// TIA Portal V19 export
DATA_BLOCK "EnS_LAcycCom_ResourceManager"   // DB39
TITLE = Instance DB of LAcycCom ResourceManager Variant
// Instance DB of LAcycCom ResourceManager Variant
// stored: InstanceOfName LAcycCom_ResourceManager_Variant, InstanceOfType FB
"LAcycCom_ResourceManager_Variant"
   // VAR_INPUT
   //    enable : Bool;
   //    config : "LAcycCom_typeResourceManagerConf";
   // END_VAR
   // VAR_OUTPUT
   //    valid : Bool;
   //    busy : Bool;
   //    error : Bool;
   //    status : Word;
   //    diagnostics : "LAcycCom_typeResourceManagerDiag";
   // END_VAR
   // VAR_IN_OUT
   //    requestBufferHeader : "LAcycCom_typeRequestBufferHeader";
   //    requestBufferElements : Variant;
   // END_VAR
   // VAR
   //    statResourceAddInfo { ExternalAccessible := 'False'; ExternalVisible := 'False'; ExternalWritable := 'False'} : Array[0..9] of Struct
   //       IOSystem : Int;
   //       station : Int;
   //    END_STRUCT;
   //    instBufferLockWatchdog { ExternalAccessible := 'False'; ExternalVisible := 'False'; ExternalWritable := 'False'; S7_SetPoint := 'True'} : TON_TIME;
   //    instRuntime { ExternalAccessible := 'False'; ExternalVisible := 'False'; ExternalWritable := 'False'; S7_SetPoint := 'True'} : TON_TIME;
   //    instCycleTime { ExternalAccessible := 'False'; ExternalVisible := 'False'; ExternalWritable := 'False'; S7_SetPoint := 'True'} : TON_TIME;
   //    instGetIMData { ExternalAccessible := 'False'; ExternalVisible := 'False'; ExternalWritable := 'False'; S7_SetPoint := 'True'} : Get_IM_Data;
   //    statIM0Data { ExternalAccessible := 'False'; ExternalVisible := 'False'; ExternalWritable := 'False'; S7_SetPoint := 'True'} : IM0_Data;
   //    statNoOfUsedResources { ExternalAccessible := 'False'; ExternalVisible := 'False'; ExternalWritable := 'False'} : Int;
   //    statUpperLimResources { ExternalAccessible := 'False'; ExternalVisible := 'False'; ExternalWritable := 'False'} : Int;
   //    statCountOfElements { ExternalAccessible := 'False'; ExternalVisible := 'False'; ExternalWritable := 'False'} : Int;
   //    statErrorUserCleared { ExternalAccessible := 'False'; ExternalVisible := 'False'; ExternalWritable := 'False'} : Bool;
   //    statErrorAutoCleared { ExternalAccessible := 'False'; ExternalVisible := 'False'; ExternalWritable := 'False'} : Bool;
   //    statEnableOld { ExternalAccessible := 'False'; ExternalVisible := 'False'; ExternalWritable := 'False'} : Bool;
   //    statDisabling { ExternalAccessible := 'False'; ExternalVisible := 'False'; ExternalWritable := 'False'} : Bool;
   // END_VAR
BEGIN
END_DATA_BLOCK
